// TIA Portal project "poke" (V16)

(* hardware
DEVICE "S71500/ET200MP station_1"  S7-1500 station
   slot 0: "导轨_0"  Rack  6ES7 590-1***0-0AA0
   slot 1: "PLC_1"  CPU 1511-1 PN  6ES7 511-1AK02-0AB0  V2.8
      slot 3: "CPU 显示_1"  6ES7591-1AA00-0AA0
      slot 32768: "PROFINET 接口_1"  X1
         slot 32769: "端口_1"  X1 P1
         slot 32770: "端口_2"  X1 P2
      slot 34817: "Virtual CP interface port_1"  Virtual CP interface port  Virtual CP interface port
*)

// ===== PLC "PLC_1"  CPU 1511-1 PN =====

VAR_GLOBAL   // PLC tag table "默认变量表"
   "Tag_1" AT %MW100 : Word;
   "Tag_2" AT %M5.0 : Bool;
   "Tag_3" AT %M5.1 : Bool;
   "m50-1" AT %M50.1 : Bool;
   "m50-2" AT %M50.2 : Bool;
   "m50-3" AT %M50.3 : Bool;
   "Clock_Byte" AT %MB0 : Byte;
   "Clock_10Hz" AT %M0.0 : Bool;
   "Clock_5Hz" AT %M0.1 : Bool;
   "Clock_2.5Hz" AT %M0.2 : Bool;
   "Clock_2Hz" AT %M0.3 : Bool;
   "Clock_1.25Hz" AT %M0.4 : Bool;
   "Clock_1Hz" AT %M0.5 : Bool;
   "Clock_0.625Hz" AT %M0.6 : Bool;
   "Clock_0.5Hz" AT %M0.7 : Bool;
   "System_Byte" AT %MB1 : Byte;
   "FirstScan" AT %M1.0 : Bool;
   "DiagStatusUpdate" AT %M1.1 : Bool;
   "AlwaysTRUE" AT %M1.2 : Bool;
   "AlwaysFALSE" AT %M1.3 : Bool;
   "m50-4" AT %M50.4 : Bool;
   "M20-0" AT %M20.0 : Bool;
   "M20-1" AT %M20.1 : Bool;
   "M20-2" AT %M20.2 : Bool;
   "MW-30" AT %MW30 : Int;
   "MD-300" AT %MD300 : DWord;
   "M20-3" AT %M20.3 : Bool;
   "M20-4" AT %M20.4 : Bool;
   "Tag_4" AT %MW400 : Int;
END_VAR

DATA_BLOCK "数据块_1"   // DB1
{ S7_Optimized_Access := 'FALSE' }
VERSION : 0.1
   VAR
      Static_1 : Pip;
      aa : Array[0..4] of Int;
   END_VAR
BEGIN
END_DATA_BLOCK

DATA_BLOCK "数据块_2"   // DB2
{ S7_Optimized_Access := 'FALSE' }
VERSION : 0.1
   VAR
      "1" : Int;
      "2" : Int;
      "3" : Int;
      "4" : Int;
      "5" : Int;
      "6" : Int;
   END_VAR
BEGIN
END_DATA_BLOCK

DATA_BLOCK "测试"   // DB3
{ S7_Optimized_Access := 'TRUE' }
VERSION : 0.1
   VAR
      地址偏移 : DInt;
      中间量 : DWord;
      循环累加 : Int;
      time1 : Time;
      add : Int;
      time2 : Time;
      time3 : Time;
      time4 : Time;
      上升沿 : Array[0..10] of Bool;
      当前时间 : Date_And_Time;
      当前时间_1 : DTL;
      当前年 : UInt;
      当前月 : UInt;
      当前日 : UInt;
      当前时 : UInt;
      当前分 : UInt;
   END_VAR
BEGIN
END_DATA_BLOCK

DATA_BLOCK "上位机温度"   // DB4
{ S7_Optimized_Access := 'FALSE' }
VERSION : 0.1
   VAR
      预热A1 : Int;
      预热A2 : Int;
      预热A3 : Int;
      预热A4 : Int;
      预热A5 : Int;
      "备用A-1" : Int;
      "备用A-2" : Int;
      "备用A-3" : Int;
      "备用A-4" : Int;
      "备用A-5" : Int;
      预热B1 : Int;
      预热B2 : Int;
      预热B3 : Int;
      预热B4 : Int;
      预热B5 : Int;
      "备用B-1" : Int;
      "备用B-2" : Int;
      "备用B-3" : Int;
      "备用B-4" : Int;
      "备用B-5" : Int;
      预热C1 : Int;
      预热C2 : Int;
      预热C3 : Int;
      预热C4 : Int;
      预热C5 : Int;
      "备用C-1" : Int;
      "备用C-2" : Int;
      "备用C-3" : Int;
      "备用C-4" : Int;
      "备用C-5" : Int;
      预热D1 : Int;
      预热D2 : Int;
      预热D3 : Int;
      预热D4 : Int;
      预热D5 : Int;
      "备用D-1" : Int;
      "备用D-2" : Int;
      "备用D-3" : Int;
      "备用D-4" : Int;
      "备用D-5" : Int;
      预热E1 : Int;
      预热E2 : Int;
      预热E3 : Int;
      预热E4 : Int;
      预热E5 : Int;
      "备用E-1" : Int;
      "备用E-2" : Int;
      "备用E-3" : Int;
      "备用E-4" : Int;
      "备用E-5" : Int;
   END_VAR
BEGIN
END_DATA_BLOCK

DATA_BLOCK "实际温度"   // DB5
{ S7_Optimized_Access := 'FALSE' }
VERSION : 0.1
   VAR
      预热A1 : Real := 500.0;
      干扰1 : Int;
      预热A2 : Real := 501.0;
      干扰2 : Int;
      预热A3 : Real := 502.0;
      干扰3 : Int;
      预热A4 : Real := 503.0;
      干扰4 : Int;
      预热A5 : Real := 504.0;
      干扰5 : Int;
      预热B1 : Real := 505.0;
      干扰6 : Int;
      预热B2 : Real := 506.0;
      干扰7 : Int;
      预热B3 : Real := 507.0;
      干扰8 : Int;
      预热B4 : Real := 508.0;
      干扰9 : Int;
      预热B5 : Real := 509.0;
      干扰10 : Int;
      预热C1 : Real := 510.0;
      干扰11 : Int;
      预热C2 : Real := 511.0;
      干扰12 : Int;
      预热C3 : Real := 512.0;
      干扰13 : Int;
      预热C4 : Real := 513.0;
      干扰14 : Int;
      预热C5 : Real := 514.0;
      干扰15 : Int;
      预热D1 : Real := 515.0;
      干扰16 : Int;
      预热D2 : Real := 516.0;
      干扰17 : Int;
      预热D3 : Real := 517.0;
      干扰18 : Int;
      预热D4 : Real := 518.0;
      干扰19 : Int;
      预热D5 : Real := 519.0;
   END_VAR
BEGIN
END_DATA_BLOCK

DATA_BLOCK "运行时间记录_DB"   // DB12
{ S7_Optimized_Access := 'TRUE' }
VERSION : 0.1
// stored: InstanceOfName 运行时间记录
"运行时间记录"
BEGIN
END_DATA_BLOCK

DATA_BLOCK "poke1"   // DB123
{ S7_Optimized_Access := 'FALSE' }
VERSION : 0.1
   VAR
      value11 : Int;
      value12 : Int;
      value13 : Int;
      value14 : Int;
      value15 : Int;
      value16 : Int;
   END_VAR
BEGIN
END_DATA_BLOCK

DATA_BLOCK "poke2"   // DB124
{ S7_Optimized_Access := 'FALSE' }
VERSION : 0.1
   VAR
      value21 : Int;
      value22 : Int;
      value23 : Int;
      value24 : Int;
      value25 : Int;
   END_VAR
BEGIN
END_DATA_BLOCK

// folder: System blocks/Program resources

DATA_BLOCK "IEC_Timer_0_DB"   // DB6
{ S7_Optimized_Access := 'TRUE' }
AUTHOR : Simatic
FAMILY : IEC
NAME : IEC_TMR
VERSION : 1.0
// stored: InstanceOfName IEC_TIMER
"IEC_TIMER"
BEGIN
END_DATA_BLOCK

DATA_BLOCK "IEC_Timer_0_DB_1"   // DB7
{ S7_Optimized_Access := 'TRUE' }
AUTHOR : Simatic
FAMILY : IEC
NAME : IEC_TMR
VERSION : 1.0
// stored: InstanceOfName IEC_TIMER
"IEC_TIMER"
BEGIN
END_DATA_BLOCK

DATA_BLOCK "IEC_Timer_0_DB_2"   // DB8
{ S7_Optimized_Access := 'TRUE' }
AUTHOR : Simatic
FAMILY : IEC
NAME : IEC_TMR
VERSION : 1.0
// stored: InstanceOfName IEC_TIMER
"IEC_TIMER"
BEGIN
END_DATA_BLOCK

DATA_BLOCK "IEC_Timer_0_DB_3"   // DB9
{ S7_Optimized_Access := 'TRUE' }
AUTHOR : Simatic
FAMILY : IEC
NAME : IEC_TMR
VERSION : 1.0
// stored: InstanceOfName IEC_TIMER
"IEC_TIMER"
BEGIN
END_DATA_BLOCK

DATA_BLOCK "IEC_Timer_0_DB_14"   // DB10
{ S7_Optimized_Access := 'TRUE' }
AUTHOR : Simatic
FAMILY : IEC
NAME : IEC_TMR
VERSION : 1.0
// stored: InstanceOfName IEC_TIMER
"IEC_TIMER"
BEGIN
END_DATA_BLOCK

DATA_BLOCK "IEC_Timer_0_DB_4"   // DB11
{ S7_Optimized_Access := 'TRUE' }
AUTHOR : Simatic
FAMILY : IEC
NAME : IEC_TMR
VERSION : 1.0
// stored: InstanceOfName IEC_TIMER
"IEC_TIMER"
BEGIN
END_DATA_BLOCK

// folder: (top level)

FUNCTION_BLOCK "11"   // FB1, LAD
{ S7_Optimized_Access := 'TRUE' }
VERSION : 0.1
   VAR CONSTANT
      "11" : Int;
   END_VAR
BEGIN
END_FUNCTION_BLOCK

FUNCTION_BLOCK "运行时间记录"   // FB2, LAD
{ S7_Optimized_Access := 'TRUE' }
VERSION : 0.1
   VAR_INPUT
      开启 : Bool;
   END_VAR
   VAR_OUTPUT
      时 : UDInt;
      分 : UDInt;
      秒 : UDInt;
   END_VAR
   VAR
      计时器 : IEC_TIMER;
      Bit位 : Array[0..10] of Bool;
   END_VAR
   VAR_TEMP   // added for the SCL form of the ladder/FBD networks
      _w1 : Bool;
   END_VAR
BEGIN

REGION Network 1
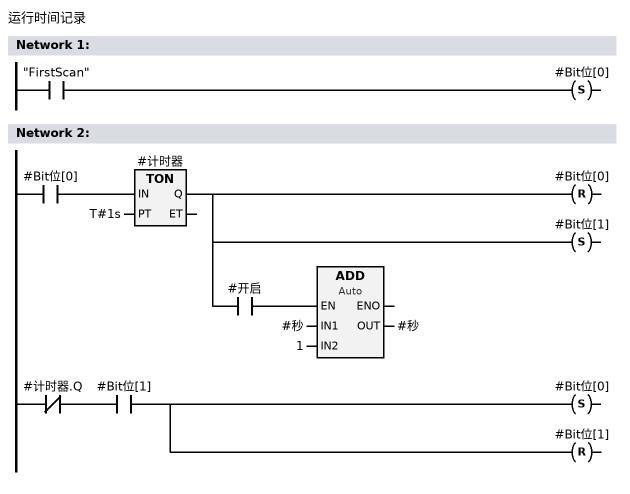
   RUNG wire#powerrail
      Contact( "FirstScan" )
      S_Coil( #Bit位[0] )
   END_RUNG
   // the same network as SCL:
   IF "FirstScan" THEN #Bit位[0] := TRUE; END_IF;
END_REGION

REGION Network 2
   #计时器.TON(IN := #Bit位[0], PT := T#1s);
   IF #计时器.Q THEN
       #Bit位[0] := FALSE;
       #Bit位[1] := TRUE;
   END_IF;
   IF #计时器.Q AND #开启 THEN #秒 := #秒 + 1; END_IF;
   #_w1 := NOT #计时器.Q AND #Bit位[1];
   IF #_w1 THEN
       #Bit位[0] := TRUE;
       #Bit位[1] := FALSE;
   END_IF;
END_REGION

REGION Network 3 (SCL)
   IF #秒 >= 60 THEN
       #分 := #分 + 1;
       #秒 := 0;
       ;
   END_IF;

   IF #分 >= 60 THEN
       #时 := #时 + 1;
       #分 := 0;
       ;
   END_IF;
END_REGION
END_FUNCTION_BLOCK

FUNCTION "循环赋值" : Bool   // FC1, LAD
{ S7_Optimized_Access := 'TRUE' }
VERSION : 0.1
   VAR_TEMP
      中间量1 : DWord;
      中间量2 : Real;
      i : Int;
      j : Int;
   END_VAR
BEGIN

REGION Network 1: 开头
END_REGION

REGION Network 2 (SCL): 测试
   //#中间量1:=PEEK_DWORD(area := 16#84, dbNumber := 5, byteOffset := 0);
   //#中间量2 := DWORD_TO_REAL(#中间量1);
   //"上位机温度".预热1 := REAL_TO_INT(#中间量2);

   //"测试".中间量 := PEEK_DWORD(area := 16#84, dbNumber := 5, byteOffset := 0);
   //"上位机温度".预热1 := DWORD_TO_INT("测试".中间量);
   // /FOR #i := 0 TO 4 DO
        #中间量1 := PEEK_DWORD(area := 16#84, dbNumber := 5, byteOffset := #i);
   //     "上位机温度".预热A1 := REAL_TO_INT(DWORD_TO_REAL(#中间量1));

   //     ;
   // END_FOR;



   //REAL_TO_INT(DWORD_TO_REAL(PEEK_DWORD(area := 16#84, dbNumber := 5, byteOffset := #i))))
   #循环赋值 := 1;
END_REGION

REGION Network 3 (SCL): 循环赋值1
   FOR #i := 0 TO 4 DO                //区域
       FOR #j := 0 TO 9 BY 2 DO             //点数
           POKE(area := 16#84,      //目标区域
                dbNumber := 4,    //目标数据块号
                byteOffset := #j + #i * 20,    //目标变量位地址 int型
                value := REAL_TO_INT((DWORD_TO_REAL(PEEK_DWORD(area := 16#84, dbNumber := 5, byteOffset := 3 * (#j + #i * 10))))));     //待写入的变量
           ;
       END_FOR;
       ;
   END_FOR;
END_REGION

REGION Network 4 (SCL): 111
   // FOR "测试".循环累加 := 0 TO 9 DO
   //     "测试".上升沿[0] := 1;
   //     "IEC_Timer_0_DB".TON(IN:="测试".上升沿[0],
   //                          PT:="测试".time1,
   //                          Q=>"测试".上升沿[0],
   //                          ET=>"测试".time2);
   //     "测试".上升沿[0] := 0;
   // END_FOR;

   IF "测试".循环累加 < 5 THEN
       "测试".上升沿[0] := 1;
       "IEC_Timer_0_DB".TON(IN := "测试".上升沿[0],
                            PT := "测试".time1,
                            Q => "测试".上升沿[1],
                            ET => "测试".time2);
       IF "测试".上升沿[1] THEN
           "IEC_Timer_0_DB_3".TON(IN := "测试".上升沿[2],
                                  PT := "测试".time3,
                                  Q => "测试".上升沿[5],
                                  ET=> "测试".time4);

           "测试".循环累加 := "测试".循环累加 + 1;
           "测试".上升沿[0] := 0;
           ;
       END_IF;

       IF "测试".循环累加 >= 5 THEN
           "测试".循环累加 := 0;
           ;
       END_IF;

       ;
   END_IF;
END_REGION
END_FUNCTION

ORGANIZATION_BLOCK "Main"   // OB1, LAD, ProgramCycle
TITLE = "Main Program Sweep (Cycle)"
{ S7_Optimized_Access := 'TRUE' }
VERSION : 0.1
   VAR_INPUT
      Initial_Call : Bool;   // Initial call of this OB
      Remanence : Bool;   // =True, if remanent data are available
   END_VAR
   VAR_TEMP   // added for the SCL form of the ladder/FBD networks
      _w1 : Bool;
      _w2 : Bool;
   END_VAR
BEGIN

REGION Network 1
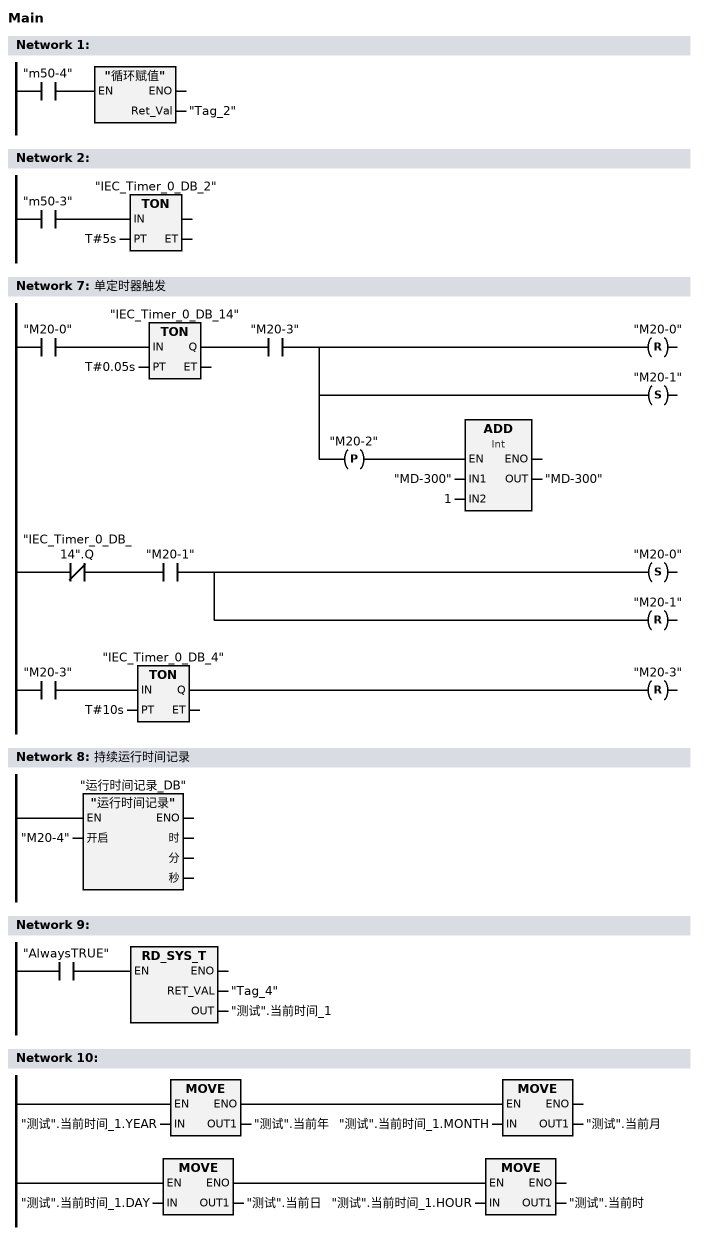
   RUNG wire#powerrail
      Contact( "m50-4" )
      "循环赋值"(Ret_Val => "Tag_2")
   END_RUNG
   // the same network as SCL:
   IF "m50-4" THEN "Tag_2" := "循环赋值"(); END_IF;
END_REGION

REGION Network 2
   "IEC_Timer_0_DB_2".TON(IN := "m50-3", PT := T#5s);
END_REGION

REGION Network 3 (SCL): POKE_BLK
   POKE_BLK(area_src := 16#84,
            dbNumber_src := 1,
            byteOffset_src := 0,
            area_dest := 16#84,
            dbNumber_dest := 2,
            byteOffset_dest := 0,
            count := 10);
END_REGION

REGION Network 4 (SCL): POKE
   POKE(area:= 16#84,      //目标区域
        dbNumber:= 123,    //目标数据块号
        byteOffset:= 8,    //目标变量位地址 int型
        value:= %DB123.DBW0 + %DB123.DBW0);     //待写入的变量
END_REGION

REGION Network 5 (SCL): peek
   "Tag_1" :=  PEEK_WORD(area := 16#84, dbNumber := 124, byteOffset := 8);
END_REGION

REGION Network 6 (SCL): 接通延时
   "IEC_Timer_0_DB_1".TON(IN := "测试".上升沿[3],
                          PT := "测试".time1,
                          Q => "测试".上升沿[4],
                          ET => "测试".time2);
END_REGION

REGION Network 7: 单定时器触发
   "IEC_Timer_0_DB_14".TON(IN := "M20-0", PT := T#0.05s);
   #_w1 := "IEC_Timer_0_DB_14".Q AND "M20-3";
   IF #_w1 THEN
       "M20-0" := FALSE;
       "M20-1" := TRUE;
   END_IF;
   #_w2 := #_w1 AND NOT "M20-2";   // rising edge
   "M20-2" := #_w1;
   IF #_w2 THEN "MD-300" := "MD-300" + 1; END_IF;
   IF NOT "IEC_Timer_0_DB_14".Q AND "M20-1" THEN
       "M20-0" := TRUE;
       "M20-1" := FALSE;
   END_IF;
   "IEC_Timer_0_DB_4".TON(IN := "M20-3", PT := T#10s);
   IF "IEC_Timer_0_DB_4".Q THEN "M20-3" := FALSE; END_IF;
END_REGION

REGION Network 8: 持续运行时间记录
   RUNG wire#powerrail
      "运行时间记录_DB"(开启 := "M20-4", 时 =>, 分 =>, 秒 =>)
   END_RUNG
   // the same network as SCL:
   "运行时间记录_DB"(开启 := "M20-4");   // "运行时间记录"
END_REGION

REGION Network 9
   IF "AlwaysTRUE" THEN "Tag_4" := RD_SYS_T(OUT => "测试".当前时间_1); END_IF;
END_REGION

REGION Network 10
   RUNG wire#powerrail
      Move(in := "测试".当前时间_1.YEAR, out1 => "测试".当前年)
      Move(in := "测试".当前时间_1.MONTH, out1 => "测试".当前月)
   END_RUNG
   RUNG wire#powerrail
      Move(in := "测试".当前时间_1.DAY, out1 => "测试".当前日)
      Move(in := "测试".当前时间_1.HOUR, out1 => "测试".当前时)
   END_RUNG
   // the same network as SCL:
   "测试".当前年 := "测试".当前时间_1.YEAR;
   "测试".当前月 := "测试".当前时间_1.MONTH;
   "测试".当前日 := "测试".当前时间_1.DAY;
   "测试".当前时 := "测试".当前时间_1.HOUR;
END_REGION
END_ORGANIZATION_BLOCK